TYPE LoggerCSV :
STRUCT
	FileSize			: ULINT;			(* (o) File size *)
	TimeCreation		: TIMESTRUCT;		(* TimeCreation of file*)
	TimeModif			: TIMESTRUCT;		(* Time Modif of file*)
	MesAlarmCode		: WORD;				(* Alarm Code*)

END_STRUCT
END_TYPE

(* stored: Version 1.1.0.1, ProductVersion 3.1.4024.6
   DUT LoggerCSV: Id {9b658292-b062-44aa-8557-bdb3ede17891} *)
